FUNCTION_BLOCK Track EXTENDS Objective IMPLEMENTS iTrack
VAR_INPUT
END_VAR
VAR_OUTPUT
END_VAR
VAR
	// TODO: hide {attribute 'hide'}
	internalOTCID			: OTCID;	// internal track id for use with MC_ActivateTrack
	internalId				: INT;	// numeric track desigination i.e. "Track 1"
END_VAR

PROPERTY Id : INT
GET
Id := internalId;
END_GET
SET
internalId := Id;
END_SET
END_PROPERTY

PROPERTY OTCID : OTCID
GET
OTCID := internalOTCID;
END_GET
SET
internalOTCID := OTCID;
END_SET
END_PROPERTY

END_FUNCTION_BLOCK

(* stored: Version 1.1.0.1, ProductVersion 3.1.4024.12
   POU Track: Id {1d568bee-17b0-45d9-8c81-c6842c2a11d5}, SpecialFunc None
   Folder Methods: Id {39635f7a-3c34-4d67-b666-c6e08a70323b}
   Folder Properties: Id {5266f954-d54f-4746-897a-a6f4b18b8998}
   Property Id: Id {bc141487-48e4-021d-1b8b-19fa2c77c46e}
   Get Get: Id {5dbdca49-4776-084f-23a4-b7b52bdccbfc}
   Set Set: Id {8e0384d9-fde2-0570-1441-0e0a49713398}
   Property OTCID: Id {6291d5a9-ab6f-0993-2dbf-1832154b326c}
   Get Get: Id {6b56faf5-f563-08e5-14ad-8b9811ab1e86}
   Set Set: Id {2e4f02ec-95b9-0171-3d64-32136881eb29} *)
